// TwinCAT 3 PLC project Samples
// ProgramVersion: 3.1.4024.0
// libraries:
//   Tc2_ControllerToolbox, * (Beckhoff Automation GmbH)
//   Tc2_EtherCAT, * (Beckhoff Automation GmbH)
//   Tc2_Standard, * (Beckhoff Automation GmbH)
//   Tc2_System, * (Beckhoff Automation GmbH)
//   Tc2_Utilities, * (Beckhoff Automation GmbH)
//   Tc3_Module, * (Beckhoff Automation GmbH)
// project tree:
//   DUTs/ ELM3002InputwTimestamp.TcDUT
//   / FasterTask.TcTTO, LEDTask.TcTTO, PlcTask.TcTTO, README.TcTLO, EventLoggerTask.TcTTO
//   POUs/Analog/ AnalogSignalProcessing.TcPOU, ToVoltageConverter.TcPOU
//   POUs/Analytics/ TimeBasedTeach.TcPOU
//   POUs/Distributed Clocks/ DistributedClockHandler.TcPOU
//   POUs/Events/DUTs/ E_EventType.TcDUT, ST_Event.TcDUT
//   POUs/Events/ EventLoggerProgram.TcPOU
//   POUs/Events/FunctionBlocks/ EventLogger.TcPOU, FB_CsvPersistentEventStorage.TcPOU
//   POUs/Events/Functions/ UpdateEventTimestampWithSystemTime.TcPOU (not stored)
//   POUs/Events/Interface/ I_PersistentEventStorage.TcIO
//   POUs/LEDs/EL2564/ Countdown.TcPOU
//   POUs/LEDs/FunctionBlocks/ LEDStateMachine.TcPOU (not stored)
//   POUs/LEDs/Functions/ RGBWToLED.TcPOU, SingleSignalToLED.TcPOU
//   POUs/LEDs/ LEDs.TcPOU
//   POUs/ MAIN.TcPOU
//   POUs/Oversampling/ OversamplingHandler.TcPOU
//   POUs/Scope/ FB_ScopeServerSample.TcPOU
//   POUs/Signal Gen/ FastSignalGen.TcPOU
//   POUs/Signal Gen/FunctionBlocks/ VariableSine.TcPOU (not stored)
//   POUs/Signal Monitoring/ SignalTimeComparison.TcPOU
//   POUs/Time/ GetDCTime.TcPOU, TimeBreakdown.TcPOU, TimerCounter.TcPOU
// real-time tasks:
//   TASK PlcTask: cycle T#1ms, priority 10, ADS port 350
//   TASK FastTask: cycle T#1ms, priority 8, ADS port 351
//   TASK FasterTask: cycle T#50us, priority 6, ADS port 352
//   TASK EventLoggerTask: cycle T#1ms, priority 12, ADS port 353
//   TASK LEDTask: cycle T#12.5us, priority 4, ADS port 354
// I/O:
//   DEVICE Device 1 (EtherCAT), AmsNetId 0.0.0.0.2.1
//     Term 5 (EK1200) [EK1200-5000 EtherCAT Power supply (2A E-Bus)]
//       Term 5 (EL2564) [EL2564 4Ch. LED output, 5...48 V DC, 4 A, RGBW]
//       Term 2 (EL4132) [EL4132 2Ch. Ana. Output +/-10V, 16bit]
//       Term 3 (ELM3002-0000) [ELM3002-0000 2Ch. Ana. Input +/-30V, 24 bit, high precision]
//       Term 9 (EL9011) [EL9011 End Terminal]
// variable links:
//   Samples/Samples Instance <-> Device 1 (EtherCAT)/Term 5 (EK1200)/Term 2 (EL4132)
//     FasterTask Outputs/FastSignalGen.voltageInv <-> Channel 2/Output
//     FasterTask Outputs/FastSignalGen.voltageOut <-> Channel 1/Output
//   Samples/Samples Instance <-> Device 1 (EtherCAT)/Term 5 (EK1200)/Term 3 (ELM3002-0000)
//     PlcTask Inputs/MAIN.oversamplingHandler.ELM3xxxSamplesIn <-> PAI Samples 20 Channel 1/Samples
//     PlcTask Inputs/MAIN.oversamplingHandler.fbDC.NextLatch <-> PAI Timestamp Channel 1/StartTimeNextLatch
//   Samples/Samples Instance <-> Device 1 (EtherCAT)/Term 5 (EK1200)/Term 5 (EL2564)
//     LEDTask Outputs/LEDs.Blue <-> PWM Outputs Channel 3/PWM output
//     LEDTask Outputs/LEDs.Green <-> PWM Outputs Channel 2/PWM output
//     LEDTask Outputs/LEDs.Red <-> PWM Outputs Channel 1/PWM output
//     LEDTask Outputs/LEDs.White <-> PWM Outputs Channel 4/PWM output

CONFIGURATION Samples
    RESOURCE PLC ON TwinCAT3
        TASK FasterTask(INTERVAL := T#50us, PRIORITY := 6);
        TASK LEDTask(INTERVAL := T#12.5us, PRIORITY := 4);
        TASK PlcTask(INTERVAL := T#1ms, PRIORITY := 10);
        TASK EventLoggerTask(INTERVAL := T#1ms, PRIORITY := 12);
        PROGRAM FastSignalGen WITH FasterTask : FastSignalGen;
        PROGRAM LEDs WITH LEDTask : LEDs;
        PROGRAM MAIN WITH PlcTask : MAIN;
        PROGRAM EventLoggerProgram WITH EventLoggerTask : EventLoggerProgram;
    END_RESOURCE
END_CONFIGURATION

// ---- DUTs/ELM3002InputwTimestamp.TcDUT
TYPE ELM3002InputwTimestamp :
STRUCT
	analogInput	:	LREAL;
	timestamp	:	ULINT;
END_STRUCT
END_TYPE

// ---- POUs/Events/DUTs/E_EventType.TcDUT
{attribute 'qualified_only'}
{attribute 'strict'}
{attribute 'to_string'}
TYPE E_EventType :
(
	Alarm := 0,
	Message := 1
);
END_TYPE

// ---- POUs/Events/DUTs/ST_Event.TcDUT
TYPE ST_Event :
STRUCT
	
	eEventType		: E_EventType;
	eEventSeverity	:	TcEventSeverity;
	nEventIdentity	:	UDINT;
	sEventText		:	STRING(255);
	dtTimestamp		:	DATE_AND_TIME;
	
END_STRUCT
END_TYPE

// ---- POUs/Events/Interface/I_PersistentEventStorage.TcIO
INTERFACE I_PersistentEventStorage

METHOD StoreEvent
VAR_INPUT
	stEvent	:	ST_Event;
END_VAR
END_METHOD

END_INTERFACE

// ---- POUs/Signal Gen/FastSignalGen.TcPOU
PROGRAM FastSignalGen
VAR
	sine	:	VariableSine;
	
	
	voltageconverter	:	ToVoltageConverter;
	
	voltageOut	AT%Q*	:	INT;
	voltageInv	AT%Q*	:	INT;
END_VAR

//sine wave generator
sine();

//sine signal to EL4132 converter
voltageconverter(in := sine.signal);
voltageOut := voltageconverter.voltage;
IF voltageOut = -32768 THEN
	voltageInv := 32767;
ELSIF voltageOut <> 0 THEN
	voltageInv := -voltageOut;
ELSE
	voltageInv := 0;
END_IF

END_PROGRAM

// ---- POUs/Analog/ToVoltageConverter.TcPOU
FUNCTION_BLOCK ToVoltageConverter
VAR_INPUT
	in	:	LREAL;
	
	negative	:	LREAL;
END_VAR
VAR_OUTPUT
	voltage	:	INT;
END_VAR
VAR
END_VAR

IF in > 0 THEN
	voltage := LREAL_TO_INT(in/10 * 32767);
ELSIF in < 0 THEN
	voltage := LREAL_TO_INT(in/10 * 32768);
ELSIF in = 0 THEN
	voltage := 0;
END_IF

END_FUNCTION_BLOCK

// ---- POUs/LEDs/LEDs.TcPOU
PROGRAM LEDs
VAR	
	Red		AT%Q*	:	INT;
	Green	AT%Q*	:	INT;
	Blue	AT%Q*	:	INT;
	White	AT%Q*	:	INT;
	
	countdown	:	Countdown;
END_VAR

countdown(RedOut => Red,GreenOut => Green, BlueOut => Blue,WhiteOut => White);

END_PROGRAM

// ---- POUs/LEDs/EL2564/Countdown.TcPOU
FUNCTION_BLOCK Countdown
VAR_INPUT
END_VAR
VAR_OUTPUT
	RedOut			:	INT;
	GreenOut		:	INT;
	BlueOut			:	INT;
	WhiteOut		:	INT;
END_VAR
VAR		
	Run		:	BOOL;
	
	ton		:	TON;
	Delay	:	TIME := T#0.5S;
	
	Countdown	:	INT		:= 5;
	On			:	BOOL	:= FALSE;;
END_VAR

// countdown to go!
IF Run THEN
	ton.IN := NOT ton.Q;
	ton.PT := Delay;
	
	IF ton.Q AND Countdown > 0 THEN //flashes 5 amber lights at < 1 second delay
		IF NOT On THEN
			RedOut := 32767;
			GreenOut := 15000;
			BlueOut := 0;
			Countdown := Countdown - 1;
			On := TRUE;
		ELSIF On THEN
			RedOut := 0;
			GreenOut := 0;
			BlueOut := 0;
			On := FALSE;
		END_IF
	ELSIF ton.Q AND Countdown = 0 THEN //go green lights 2 second delay
		GreenOut := 32767;
		RedOut := 0;
		BlueOut := 0;
		Countdown := -1;
	ELSIF ton.Q AND Countdown < 0 THEN //turns off countdown and resets counter after 2 seconds of green
		Run := FALSE;
		RedOut := 0;
		GreenOut := 0;
		BlueOut := 0;
	END_IF
	
	IF Countdown = 0 THEN
		Delay := T#2S;
	END_IF
	
	ton();
ELSIF NOT Run THEN
	RedOut := 0;
	GreenOut := 0;
	BlueOut := 10000;
	WhiteOut := 0;
	Countdown := 5;
	Delay := T#0.5S;
END_IF

END_FUNCTION_BLOCK

// ---- POUs/MAIN.TcPOU
PROGRAM MAIN
VAR		
	bRun	:	BOOL := FALSE;
	
	secondtimer	:	TimerCounter;
	
	oversamplingHandler	:	OversamplingHandler;
	
	//EL3751 signals in
	voltageIn	AT%I*	:	DINT;
	voltageIn2	AT%I*	:	DINT;
	
	EL3xxx	:	AnalogSignalProcessing;
	ELM3xxx	:	AnalogSignalProcessing;
	
	primaryVoltage		: LREAL;
	secondaryVoltage	:	LREAL;
	
	//scope server control block
(*	fbScopeServer	:	FB_ScopeServerSample;
	xStartStopScope	:	BOOL;
	*)
	
	//Analytics Teach FB
	//fbTimeTeach	:	TimeBasedTeach;
	
	// dc time stuff
	fbSystemDCTime	:	GetDCTime;
END_VAR

IF bRun THEN
		
	//Timer counter fb
	//secondtimer();
	
	//oversampling - ELM3002 processing
	oversamplingHandler();
	
	//EL3751 reading signal
	(*EL3xxx(signalIn := voltageIn);
	ELM3xxx(signalIn := voltageIn2);*)
	
	//EL3751 Signal processing
	//primaryVoltage := EL3xxx.voltageIn;
	//secondaryVoltage := ELM3xxx.voltageIn;
	
	//Scope server control from PLC
	(*
	fbScopeServer(
		sNetId					:='5.119.159.52.1.1', 
		bExternalTriggerEvent	:=xStartStopScope , 
		sConfigFile				:= 'C:\Y.tcscopex', 
		sSaveFile				:='C:\Record.svdx' , 
		bBusy					=> , 
		bError					=>, 
		nErrorId				=>);
	*)
	
	//fbTimeTeach();

	fbSystemDCTime();
	
END_IF

bRun := True;

END_PROGRAM

// ---- POUs/Time/TimerCounter.TcPOU
FUNCTION_BLOCK TimerCounter
VAR
	bRun	AT%I*	:	BOOL;
	bTest	AT%Q*	:	BOOL;
	iCounter	AT%Q*	:	INT;
	
	ton		:	TON;
END_VAR

IF bRun THEN
	ton.IN := NOT ton.Q;
	ton.PT := T#1S;
	
	IF ton.Q THEN
		iCounter := iCounter + 1;
		bTest := NOT bTest;
	END_IF
	
	IF iCounter > 10000 THEN
		iCounter := 0;
	END_IF
	
	ton();
END_IF

END_FUNCTION_BLOCK

// ---- POUs/Oversampling/OversamplingHandler.TcPOU
FUNCTION_BLOCK OversamplingHandler
VAR_INPUT
END_VAR
VAR_OUTPUT
END_VAR
VAR
	i	:	INT;
	
	ELM3xxxSamplesIn	AT%I*	:	ARRAY[0..noOfSamples] OF DINT;
	ELM3xxxSamplesOut	:	ARRAY[0..noOfSamples] OF LREAL;
	
	PM10VMax	:	LREAL := 7812500; //8388607 - 24bit not extended
	PM10VMin	:	LREAL := 7812500;
	PM10Mult	:	LREAL := 10;
	
	fbSignal	:	SignalTimeComparison;
	
	fbDC	:	DistributedClockHandler;
END_VAR
VAR CONSTANT
	noOfSamples	:	INT := 19;
END_VAR

FOR i := 0 TO noOfSamples DO
	ELM3xxxSamplesOut[i] := AnalogSignalConverter(input := ELM3xxxSamplesIn[i], maximum := PM10VMax, minimum := PM10VMin, multiplier := PM10Mult);
END_FOR

fbDC(Samples := ELM3xxxSamplesOut);

METHOD AnalogSignalConverter : LREAL
VAR_INPUT
	input		:	LREAL;
	maximum		:	LREAL;
	minimum		:	LREAL;
	multiplier	:	LREAL;
END_VAR
IF input > 0 THEN
	AnalogSignalConverter := (input/maximum) * multiplier;
ELSIF input < 0 THEN
	AnalogSignalConverter := (input/minimum) * multiplier;
ELSIF input = 0 THEN
	AnalogSignalConverter := 0;
END_IF
END_METHOD

END_FUNCTION_BLOCK

// ---- POUs/Signal Monitoring/SignalTimeComparison.TcPOU
FUNCTION_BLOCK SignalTimeComparison
VAR_INPUT
	insignalTime	:	ULINT;
	outsignalTime	:	ULINT;
END_VAR
VAR_OUTPUT
	seconds	:	ULINT;
	milseconds	:	ULINT;
	micseconds	:	ULINT;
	nseconds	:	ULINT;
END_VAR
VAR
END_VAR
VAR CONSTANT
	noOfSamples	:	INT := 19;
END_VAR

nseconds := (insignalTime MOD 1000) - (outsignalTime MOD 1000);

micseconds := ((insignalTime MOD 1000000) - (outsignalTime MOD 1000000))/1000;

milseconds := ((insignalTime MOD 1000000000) - (outsignalTime MOD 1000000000))/1000000;

seconds := (insignalTime/1000000000) - (outsignalTime/1000000000);

END_FUNCTION_BLOCK

// ---- POUs/Distributed Clocks/DistributedClockHandler.TcPOU
FUNCTION_BLOCK DistributedClockHandler
VAR_INPUT	
	Samples	:	ARRAY[0..noOfSamples] OF LREAL;
END_VAR
VAR_OUTPUT
END_VAR
VAR
	TimeBreakdown	:	TimeBreakdown;

	NextLatch	AT%I*	:	ULINT;
	CurrentLatch	:	ULINT;
	
	Timestamps	:	ARRAY[0..noOfSamples] OF ULINT;
	
END_VAR
VAR CONSTANT
	noOfSamples		:	INT		:= 19;
END_VAR

IF CurrentLatch <> 0 THEN
	CalculateTimestamps();
END_IF

CurrentLatch := NextLatch;

METHOD CalculateTimestamps
VAR
	sampleIterator	:	INT;
END_VAR
VAR CONSTANT
	cycleTime		:	ULINT	:= 1000000;
	sampleDistance	:	UINT	:= 50000;
END_VAR
FOR sampleIterator := 0 TO noOfSamples DO
	Timestamps[sampleIterator] := (CurrentLatch - cycleTime) - (INT_TO_ULINT(sampleIterator) * sampleDistance);
END_FOR
END_METHOD

END_FUNCTION_BLOCK

// ---- POUs/Time/TimeBreakdown.TcPOU
FUNCTION_BLOCK TimeBreakdown
VAR_INPUT
	timesignal	:	ULINT;
END_VAR
VAR_OUTPUT	
	seconds	:	ULINT;
	milseconds	:	ULINT;
	micseconds	:	ULINT;
	nseconds	:	ULINT;
END_VAR
VAR	
END_VAR

nseconds := timesignal MOD 1000;

micseconds := (timesignal MOD 1000000)/1000;

milseconds := (timesignal MOD 1000000000)/1000000;

seconds := (timesignal MOD 1000000000000)/1000000000;

END_FUNCTION_BLOCK

// ---- POUs/Analog/AnalogSignalProcessing.TcPOU
FUNCTION_BLOCK AnalogSignalProcessing
VAR_INPUT
	signalIn	:	DINT;
END_VAR
VAR_OUTPUT
END_VAR
VAR
	PM10VMax	:	LREAL := 7812500; //8388607 - 24bit not extended
	PM10VMin	:	LREAL := 7812500;
	PM10Mult	:	LREAL := 10;
	
	voltageIn	:	LREAL;
END_VAR

voltageIn := AnalogSignalConverter(input := signalIn, maximum := PM10VMax, minimum := PM10VMin, multiplier := PM10Mult);

METHOD AnalogSignalConverter : LREAL
VAR_INPUT
	input		:	LREAL;
	maximum		:	LREAL;
	minimum		:	LREAL;
	multiplier	:	LREAL;
END_VAR
IF input > 0 THEN
	AnalogSignalConverter := (input/maximum) * multiplier;
ELSIF input < 0 THEN
	AnalogSignalConverter := (input/minimum) * multiplier;
ELSIF input = 0 THEN
	AnalogSignalConverter := 0;
END_IF
END_METHOD

END_FUNCTION_BLOCK

// ---- POUs/Time/GetDCTime.TcPOU
FUNCTION_BLOCK GetDCTime
VAR_INPUT
END_VAR
VAR_OUTPUT
	actual	:	ULINT;
	tasktime	:	ULINT;
	ticktime	:	ULINT;
END_VAR
VAR
	aminustask	:	ULINT;
	aminustick	:	ULINT;
	taskminustick	:	ULINT;
	
	bb	:	BOOL;
	
	signalcomp :	SignalTimeComparison;
END_VAR

actual := F_GetActualDcTime64();
tasktime := F_GetCurDcTaskTime64();
ticktime := F_GetCurDcTickTime64();


// compares the offset to different dc time functions
IF bb THEN
	aminustask := actual - tasktime;
	aminustick := actual - ticktime;
	taskminustick := tasktime - ticktime;
	
	signalcomp(insignalTime := actual, outsignalTime := tasktime);
	
	bb := FALSE;
END_IF

END_FUNCTION_BLOCK

// ---- POUs/Events/EventLoggerProgram.TcPOU
PROGRAM EventLoggerProgram
VAR
	bBoolean	:	BOOL;	

	eEventType		: E_EventType := E_EventType.Alarm;
	eEventSeverity	:	TcEventSeverity := TcEventSeverity.Error;
	nEventIdentity	:	UDINT := 42;
	sEventText		:	STRING(255) := 'An Error has occured';
	
	CsvPersistentEventStorage	:	FB_CsvPersistentEventStorage;
	EventLogger	:	EventLogger(CsvPersistentEventStorage);
END_VAR

IF bBoolean THEN
	EventLogger.AddEvent(eEventType, eEventSeverity, nEventIdentity, sEventText);	
	bBoolean := FALSE;
END_IF

CsvPersistentEventStorage();

END_PROGRAM

// ---- POUs/Events/FunctionBlocks/FB_CsvPersistentEventStorage.TcPOU
FUNCTION_BLOCK FB_CsvPersistentEventStorage IMPLEMENTS I_PersistentEventStorage //Functionality only allows for one event added per cycle, implementation of more requires a buffer
VAR
	stEventWrittenToFile	:	ST_Event;
	
	fbFileOpen	:	FB_FileOpen	:= (sPathName := 'C:\Events.log', nMode := FOPEN_MODEAPPEND OR FOPEN_MODETEXT);
	fbFilePuts	:	FB_FilePuts;	
	fbFileClose	:	FB_FileClose;
	
	CsvString	:	T_MaxString;
	
	eWriteState	:	(FILE_OPEN_TRIGGER, FILE_OPEN, WAIT_FOR_EVENT, WRITE_EVENT_TRIGGER, WRITE_EVENT, FILE_CLOSE_TRIGGER, FILE_CLOSE, ERROR);
	
	EventBuffer	:	ARRAY[0..99] OF ST_Event;
	CurrentEventBufferIndex	:	INT	:=	0;
	EventsWritten	:	INT	:= 0;
END_VAR
VAR CONSTANT
	MAXIMUM_SIZE_OF_EVENT_BUFFER	:	INT := 99;
END_VAR

IF NOT (CurrentEventBufferIndex = EventsWritten) AND eWriteState <> WAIT_FOR_EVENT  THEN
	stEventWrittenToFile := EventBuffer[EventsWritten];
	CsvWrite(stEventWrittenToFile);
END_IF

METHOD PRIVATE CreateCsvString : T_MaxString
VAR_INPUT
	stEvent	:	REFERENCE TO ST_Event;
END_VAR
VAR
	TempString	:	T_MaxString;
END_VAR
TempString := TO_STRING(stEvent.eEventType);
TempString := CONCAT(STR1 := TempString, STR2 := ',');
TempString := CONCAT(STR1 := TempString, STR2 := TO_STRING(stEvent.eEventSeverity));
TempString := CONCAT(STR1 := TempString, STR2 := ',');
TempString := CONCAT(STR1 := TempString, STR2 := TO_STRING(stEvent.nEventIdentity));
TempString := CONCAT(STR1 := TempString, STR2 := ',');
TempString := CONCAT(STR1 := TempString, STR2 := stEvent.sEventText);
TempString := CONCAT(STR1 := TempString, STR2 := ',');
TempString := CONCAT(STR1 := TempString, STR2 := TO_STRING(stEvent.dtTimestamp));
TempString := CONCAT(STR1 := TempString, STR2 := '$n');

CreateCsvString := TempString;
END_METHOD

METHOD CsvWrite
VAR_INPUT
	stEventBeingWritten	:	ST_Event;
END_VAR
CASE eWriteState OF
	FILE_OPEN_TRIGGER:
		fbFileOpen(bExecute := TRUE);
		eWriteState := FILE_OPEN;
	
	FILE_OPEN:
		fbFileOpen(bExecute := FALSE);
		IF fbFileOpen.bError THEN
			eWriteState := ERROR;
		ELSIF NOT fbFileOpen.bError AND fbFileOpen.hFile <> 0 THEN
			eWriteState := WRITE_EVENT_TRIGGER;
		END_IF
		
	WRITE_EVENT_TRIGGER:
		CsvString := CreateCsvString(stEvent := stEventBeingWritten);
		fbFilePuts(bExecute := TRUE, 
					sLine := CsvString, 
					hFile := fbFileOpen.hFile);
		eWriteState := WRITE_EVENT;
	
	WRITE_EVENT:
		fbFilePuts(bExecute := FALSE);
		IF fbFilePuts.bError THEN
			eWriteState := ERROR;
		ELSIF NOT fbFilePuts.bError THEN
			EventsWritten := EventsWritten + 1;
			eWriteState := FILE_CLOSE_TRIGGER;
		END_IF

	FILE_CLOSE_TRIGGER:
		fbFileClose(bExecute := TRUE, hFile := fbFileOpen.hFile);
		eWriteState := FILE_CLOSE;
		
	FILE_CLOSE:
		fbFileClose(bExecute := FALSE);
		IF fbFileClose.bError THEN
			eWriteState := ERROR;
		ELSIF NOT fbFileClose.bError THEN
			eWriteState := WAIT_FOR_EVENT;
		END_IF
		
	WAIT_FOR_EVENT:
	// Do nothing

	ERROR:
	// Do nothing

END_CASE
END_METHOD

METHOD IsEventBufferFull : BOOL
VAR_INPUT
END_VAR
IF (CurrentEventBufferIndex + 1) > MAXIMUM_SIZE_OF_EVENT_BUFFER THEN
	IsEventBufferFull := TRUE;
END_IF
END_METHOD

METHOD StoreEvent
VAR_INPUT
	stEvent	: ST_Event;
END_VAR
IF NOT IsEventBufferFull() THEN
	EventBuffer[CurrentEventBufferIndex] := stEvent;
	CurrentEventBufferIndex := CurrentEventBufferIndex + 1;
	eWriteState := FILE_OPEN_TRIGGER;
END_IF
END_METHOD

END_FUNCTION_BLOCK

// ---- POUs/Events/FunctionBlocks/EventLogger.TcPOU
FUNCTION_BLOCK EventLogger 
VAR
	EventBuffer	:	ARRAY[1..100] OF ST_Event; // Stores events, event buffer
	CurrentEventBufferIndex	:	INT := 0;
	
	_PersistentEventStorage	:	I_PersistentEventStorage;
END_VAR
VAR CONSTANT
	MAXIMUM_SIZE_OF_EVENT_BUFFER	:	INT := 100;
END_VAR

(* True for successful add, false for full buffer*)
METHOD PUBLIC AddEvent : BOOL
VAR_INPUT
	eEventType		: E_EventType;
	eEventSeverity	:	TcEventSeverity;
	nEventIdentity	:	UDINT;
	sEventText		:	STRING(255);
END_VAR
IF NOT IsEventBufferFull() THEN
	CurrentEventBufferIndex := CurrentEventBufferIndex + 1;
	EventBuffer[CurrentEventBufferIndex].eEventType := eEventType;
	EventBuffer[CurrentEventBufferIndex].eEventSeverity := eEventSeverity;
	EventBuffer[CurrentEventBufferIndex].nEventIdentity := nEventIdentity;
	EventBuffer[CurrentEventBufferIndex].sEventText := sEventText;
	UpdateEventTimestampWithSystemTime(stEvent := EventBuffer[CurrentEventBufferIndex]);

	AddEvent := TRUE;
ELSE
	AddEvent := FALSE;
END_IF

// store event persistently
_PersistentEventStorage.StoreEvent(stEvent := EventBuffer[CurrentEventBufferIndex]);
END_METHOD

METHOD FB_Init : BOOL
VAR_INPUT
	bInitRetains	:	BOOL; // if true, retain variables are initialised (warm / cold start)
	bInCopyCode		:	BOOL; // if true, instance after gets moved into the copy code (online change)
	iPersistentEventStorage		:	I_PersistentEventStorage;
END_VAR
_PersistentEventStorage := iPersistentEventStorage;
END_METHOD

METHOD IsEventBufferFull : BOOL
VAR_INPUT
END_VAR
IF (CurrentEventBufferIndex + 1) > MAXIMUM_SIZE_OF_EVENT_BUFFER THEN
	IsEventBufferFull := TRUE;
END_IF
END_METHOD

END_FUNCTION_BLOCK

// ---- POUs/Analytics/TimeBasedTeach.TcPOU
FUNCTION_BLOCK TimeBasedTeach
VAR_INPUT
END_VAR
VAR_OUTPUT
END_VAR
VAR
	bStartTeach	AT%I*	:	BOOL;
	bStopTeach	AT%Q*	:	BOOL;
	
	ton	:	TON;
END_VAR

IF bStartTeach THEN
	ton.IN := NOT ton.Q;
	ton.PT := T#5S;
	
	//ensure StopTeach is False
	bStopTeach := FALSE;
	
	IF ton.Q THEN
		bStartTeach := FALSE;
		bStopTeach := TRUE;
	END_IF
END_IF

END_FUNCTION_BLOCK

// ---- POUs/LEDs/Functions/RGBWToLED.TcPOU
FUNCTION RGBWToLED
VAR_INPUT
	RedIn	:	USINT;
	GreenIn	:	USINT;
	BlueIn	:	USINT;
	WhiteIn	:	USINT;
END_VAR
VAR_OUTPUT
	RedOut		:	INT;
	GreenOut	:	INT;
	BlueOut		:	INT;
	WhiteOut	:	INT;
END_VAR

RedOut := SingleSignalToLED(RedIn);
GreenOut := SingleSignalToLED(GreenIn);
BlueOut := SingleSignalToLED(BlueIn);
WhiteOut := SingleSignalToLED(WhiteIn);

END_FUNCTION

// ---- POUs/LEDs/Functions/SingleSignalToLED.TcPOU
FUNCTION SingleSignalToLED : INT
VAR_INPUT
	LEDSignal	:	USINT;
END_VAR
VAR
END_VAR

// convert standard 0-255 LED signals to INT datatype
SingleSignalToLED := LEDSignal/256 * 32767;

END_FUNCTION

// ---- POUs/Scope/FB_ScopeServerSample.TcPOU
FUNCTION_BLOCK FB_ScopeServerSample
VAR_INPUT
	sNetId					: STRING	:='';	
    bExternalTriggerEvent	: BOOL 		:= FALSE; //Rising edge start recording, falling edge stop and save
	sConfigFile				: STRING(80); //.tcscopex
	sSaveFile				: STRING(80); //.svdx
END_VAR
VAR_OUTPUT
    bBusy					: BOOL 		:= FALSE;
    bError					: BOOL 		:= FALSE;
    nErrorId				: UDINT 	:= 0;	
END_VAR
VAR

    bDone					: BOOL 		:= FALSE;	

    fbScopeServerControl	: FB_ScopeServerControl;
    eReqState				: E_ScopeServerState := SCOPE_SERVER_IDLE;
	
    eState					: (IDLE,RECORDING,SAVING,DISCONNECTING,ERROR,RESETING);
END_VAR

CASE eState OF
	IDLE:
		bBusy	:=FALSE;
		IF bExternalTriggerEvent THEN
			bBusy			:= TRUE;
	    	eReqState 		:= SCOPE_SERVER_START;
	    	eState 			:= RECORDING;	
		END_IF
	
	RECORDING:	
		IF fbScopeServerControl.bDone THEN
	    	IF NOT bExternalTriggerEvent THEN
	    	    eReqState 		:= SCOPE_SERVER_SAVE;
	    	    eState 			:= SAVING;
	    	END_IF
		ELSIF fbScopeServerControl.bError THEN
			eState	:=ERROR;		
		END_IF
		
	SAVING:
	    IF fbScopeServerControl.bDone THEN
	        eReqState 		:= SCOPE_SERVER_DISCONNECT;
			eState			:= DISCONNECTING;
		ELSIF fbScopeServerControl.bError THEN
			eState	:=ERROR;		
		END_IF
		
	DISCONNECTING:
		IF fbScopeServerControl.bDone THEN
	       eState := IDLE;
		ELSIF fbScopeServerControl.bError THEN
			eState	:=ERROR;				   
	    END_IF		
		
	ERROR:
		bBusy			:= FALSE;
		IF NOT bExternalTriggerEvent THEN
			bBusy			:= TRUE;
			eReqState 		:= SCOPE_SERVER_RESET;
			eState			:= DISCONNECTING;
		END_IF
		
	RESETING:
		IF fbScopeServerControl.bDone OR fbScopeServerControl.bError THEN
	       	eReqState 		:= SCOPE_SERVER_IDLE;
			eState			:= IDLE; 
	    END_IF		
		
END_CASE


fbScopeServerControl( sNetId		:= '5.119.159.52.1.1',
                      eReqState		:= eReqState,
                      sConfigFile	:= sConfigFile,
                      sSaveFile		:= sSaveFile,
                      tTimeout		:= T#2S,
                      bBusy			=>,
                      bDone			=>bDone,
                      bError		=>bError,
                      nErrorId		=>nErrorId);

END_FUNCTION_BLOCK

// ---- README.TcTLO
TEXTLIST README
  TestInProgress is for testing new features, MAIN is for developing test code = ''
   = ''
END_TEXTLIST
